{attribute 'qualified_only'}
//{attribute 'strict'}
TYPE E_TrackNum :
(
	Big		:=1,
	Small	:=2,
	Main	:=3
);	
END_TYPE

(* stored: Version 1.1.0.1
   DUT E_TrackNum: Id {8c7b446a-e63b-4ff3-8581-b59315de87a2} *)
